// TwinCAT 3 PLC project Simulatore_ASRV
// ProgramVersion: 3.1.4023.0
// libraries:
//   Tc2_Standard, * (Beckhoff Automation GmbH)
//   Tc2_System, * (Beckhoff Automation GmbH)
//   Tc2_Utilities, * (Beckhoff Automation GmbH)
//   Tc3_Module, * (Beckhoff Automation GmbH)
//   VisuDialogs, * (System)
//   VisuSymbols,3.5.10.0,System
// project tree:
//   DUTs/ ASRV.TcDUT, RX_CMD_PC.TcDUT, Comando_PC.TcDUT, CMD_PC.TcDUT, RX_MIS_PC.TcDUT, MIS_PC.TcDUT, Stato_ASRV.TcDUT, Stato_Aux_ASRV.TcDUT, Comandi.TcDUT, Step_PC.TcDUT, RX_Step_PC.TcDUT, TX_STA_ASRV.TcDUT, STA_ASRV.TcDUT
//   / Gestore di visualizzazione.TcVMO (not stored), GlobalTextList.TcGTLO, PlcTask.TcTTO, VISU_TASK.TcTTO
//   GVLs/ Var_Globali.TcGVL
//   POUs/ Check_Com_PC.TcPOU, FB_ClassASRV.TcPOU, FB_File_Write.TcPOU, FB_File_Read.TcPOU, MAIN.TcPOU, Simula_Compila_Mis.TcPOU, Simula_Compila_Sta.TcPOU, Reset_Mis.TcPOU, Simula_Run_Mis.TcPOU, FB_Test_XXX.TcPOU, Trasf_Sta_TxSta.TcPOU, Trasf_RxMiss_Miss.TcPOU, Trasf_RxCmd_Cmd.TcPOU
//   VISUs/ Visualization.TcVIS
// real-time tasks:
//   TASK PlcTask: cycle T#10ms, priority 6, ADS port 350
//   TASK VISU_TASK: cycle T#100000us, priority 8, ADS port 351

CONFIGURATION Simulatore_ASRV
    RESOURCE PLC ON TwinCAT3
        TASK PlcTask(INTERVAL := T#10ms, PRIORITY := 6);
        TASK VISU_TASK(INTERVAL := T#100000us, PRIORITY := 8);
        PROGRAM MAIN WITH PlcTask : MAIN;
        PROGRAM VisuElems_Visu_Prg WITH VISU_TASK : VisuElems.Visu_Prg;
    END_RESOURCE
END_CONFIGURATION

// ---- DUTs/ASRV.TcDUT
TYPE ASRV :
STRUCT
	ASRV_MIS 	: MIS_PC;		// missione da PC
	ASRV_CMD	: CMD_PC;		// comandi da PC
	ASRV_STA	: STA_ASRV;		// stato ASRV
	ASRV_num 	: UINT;			// numero ASRV
END_STRUCT
END_TYPE

// ---- DUTs/RX_CMD_PC.TcDUT
TYPE RX_CMD_PC :
STRUCT
	WatchDog_PC        : UINT;  		// Check di rete (PC++, ASRV pareggia) 
	Start_Miss_PC      : UINT;			// Start Missione da PC. Start=1, azzera appena Stato_Miss_ASRV=1
	End_Miss_PC        : UINT;			// Fine Missione da PC. End=1, appena Stato_Miss_ASRV=2 o per forz.PC
	Pintend_PC         : UINT;			// Nodo intermedio missione = Nodo semaforo di stop
	New_Pos_PC         : UINT;			// Nodo assegnato da PC a ASRV
	Comando_PC         : WORD;			// Word (16 bit) --> struttura Comando PC (16 byte)			
END_STRUCT
END_TYPE

// ---- DUTs/Comando_PC.TcDUT
TYPE Comando_PC :
STRUCT
	Stop    : BOOL; 	// Arresta ASRV immediatamente 
	Aux1	: BOOL;			
	Aux2	: BOOL;			
	Aux3	: BOOL;			
	Aux4	: BOOL;			
	Aux5	: BOOL;			
	Aux6	: BOOL;			
	Aux7	: BOOL;			
	Aux8	: BOOL;			
	Aux9	: BOOL;			
	Aux10	: BOOL;			
	Aux11	: BOOL;			
	Aux12	: BOOL;			
	Aux13	: BOOL;			
	Aux14	: BOOL;			
	Aux15	: BOOL;			
 END_STRUCT
END_TYPE

// ---- DUTs/CMD_PC.TcDUT
TYPE CMD_PC :
STRUCT
	WatchDog_PC        : UINT;  		// Check di rete (ASRV++, PC pareggia) 
	Start_Miss_PC      : UINT;			// Start Missione da PC. Start=1, azzera appena Stato_Miss_ASRV=1
	End_Miss_PC        : UINT;			// Fine Missione da PC. End=1, appena Stato_Miss_ASRV=2 o per forz.PC
	Pintend_PC         : UINT;			// Nodo intermedio missione = Nodo semaforo di stop
	New_Pos_PC         : UINT;			// Nodo assegnato da PC a ASRV
	Comando_PC         : Comando_PC;	// struttura Comando PC			
END_STRUCT
END_TYPE

// ---- DUTs/RX_MIS_PC.TcDUT
TYPE RX_MIS_PC :
STRUCT
	Step_PC       : ARRAY[0..MAX_STEP_MISS] OF RX_Step_PC; // Word ==> step programma 0..500
	Tot_step_PC	  : UINT;						 // Numero di steps della missione
	Pstart_PC     : UINT;						 // Nodo iniziale missione (=Nodo attuale ASRV)
	Pend_PC       : UINT;						 // Nodo fine missione (eventuale di carico/scarico)
	Typ_car_PC    : UINT;						 // Tipo di stabilità carico (0 massima, 9 minima)
	MisFree1      : UINT;
	MisFree2      : UINT;
	MisFree3      : UINT;
END_STRUCT
END_TYPE

// ---- DUTs/MIS_PC.TcDUT
TYPE MIS_PC :
STRUCT
	Step_PC       : ARRAY[0..MAX_STEP_MISS] OF Step_PC;	// Array step programma  (0..500)
	Tot_step_PC	  : UINT;						// Numero di steps della missione
	Pstart_PC     : UINT;						// Nodo iniziale missione (=Nodo attuale ASRV)
	Pend_PC       : UINT;						// Nodo fine missione (eventuale di carico/scarico)
	Typ_car_PC    : UINT;						// Tipo di stabilità carico (0 massima, 9 minima)
	MisFree1      : UINT;
	MisFree2      : UINT;
	MisFree3      : UINT;
END_STRUCT
END_TYPE

// ---- DUTs/Stato_ASRV.TcDUT
TYPE Stato_ASRV :
STRUCT
	In_Mov_X      : BOOL;	// In movimento su asse X (orizz)
	In_Mov_Y      : BOOL;	// In movimento su asse Y (vert)
	In_Mov_Av     : BOOL;	// In movimento direzione +
	In_Mov_Ind    : BOOL;	// In movimento direzione -
	In_Allarme    : BOOL;	// In allarme
	Ok_Prog       : BOOL;	// Pronto a ricevere Missione
	In_Automatico : BOOL;	// In Automatico
	In_Manuale    : BOOL;	// In Manuale	
	Su_Nodo       : BOOL;	// Posizionato su Nodo
	Carico        : BOOL;	// Pallet a bordo
	PosSoll_0     : BOOL;	// Codifica pos. alzata pallet bit.0
	PosSoll_1     : BOOL;	// Codifica pos. alzata pallet bit.1
	Rich_Reset    : BOOL;	// Richiede reset missione a Supervisore
	Aux13         : BOOL;
	Aux14         : BOOL;
	Aux15         : BOOL;
END_STRUCT
END_TYPE

// ---- DUTs/Stato_Aux_ASRV.TcDUT
TYPE Stato_Aux_ASRV :
STRUCT
	Fermo_in_X    : BOOL;	// Fermo su asse X (orizz)
	Fermo_in_Y    : BOOL;	// Fermo su asse Y (vert)
	Rotaz_in_X    : BOOL;	// In rotazione verso asse X
	Rotaz_in_y    : BOOL;	// In rotazione verso asse X
	In_Ricarica   : BOOL;	// In ricarica batteria
	In_Sost_Batt  : BOOL;	// In sostituzione batteria
	In_Manutenz   : BOOL;	// In manutenzione
	Aux7          : BOOL;		
	Aux8          : BOOL;	
	Aux9          : BOOL;	
	Aux10         : BOOL;	
	Aux11         : BOOL;	
	Aux12         : BOOL;	
	Aux13         : BOOL;
	Aux14         : BOOL;
	Aux15         : BOOL;
END_STRUCT
END_TYPE

// ---- DUTs/Comandi.TcDUT
TYPE Comandi :
STRUCT
	In_Mov_X    : BOOL;		// Muovi su asse X
	In_Mov_Y    : BOOL;		// Muovi su asse Y
	In_Mov_Av   : BOOL;		// Muovi direzione +
	In_Mov_Ind  : BOOL;		// Muovi direzione -
	CarSoll_0   : BOOL;		// Carica pallet (codice alza pallet bit 0)
	CarSoll_1   : BOOL;		// Carica pallet (codice alza pallet bit 1)
	Scarica     : BOOL;		// Scarica pallet
	Lenta       : BOOL;		// Muovi in lenta
	End         : BOOL;		// Fine Missione (ultimo step)
	Aux9		: BOOL;		
	Aux10		: BOOL;	
	Aux11		: BOOL;
	Aux12		: BOOL;
	Aux13		: BOOL;
	Aux14		: BOOL;
	Aux15		: BOOL;
END_STRUCT
END_TYPE

// ---- DUTs/Step_PC.TcDUT
TYPE Step_PC :
STRUCT
	Comandi      : Comandi;
	ps		     : UINT;		// Nodo da raggiungere nello step
	dist	     : UINT;		// Distanza del Nodo da raggiungere (in cm)
	rall	     : UINT;		// Rallentamento speccifico nello Step
	CmFree1		 : UINT;		
	CmFree2		 : UINT;		
	CmFree3		 : UINT;		
END_STRUCT
END_TYPE

// ---- DUTs/RX_Step_PC.TcDUT
TYPE RX_Step_PC :
STRUCT
	Comandi      : WORD;		// Word (16 bit) ==> comandi (16 byte)
	ps		     : UINT;		// Nodo da raggiungere nello step
	dist	     : UINT;		// Distanza del Nodo da raggiungere (in cm)
	rall	     : UINT;		// Rallentamento specifico nello Step
	CmFree1		 : UINT;		
	CmFree2		 : UINT;		
	CmFree3		 : UINT;		
END_STRUCT
END_TYPE

// ---- DUTs/TX_STA_ASRV.TcDUT
TYPE TX_STA_ASRV :
STRUCT
	WatchDog_ASRV        : UINT;  			// Check di rete (ASRV++, PC pareggia) 
	Pos_ASRV             : UINT; 	    	// Nodo attuale ASRV
	Stato_Miss_ASRV      : UINT;			// Stato Missione ASRV (0=idle, 1=attiva, 2=completa)
	Stato_ASRV           : WORD;		    // Word (16 bit) ==> struct Stato_ASRV (16 byte)
	Stato_Aux_ASRV 	     : WORD;		 	// Word (16 bit) ==> struct Stato_Aux_ASRV (16 byte)
	ptr_step_ASRV	     : UINT;			// Puntatore passo programma (in esecuzione)
	offset_da_nodo_ASRV  : UINT;			// distanza da ultimo Nodo (in cm)
	Allarmi_1_ASRV       : WORD;			// allarmi ASRV word 1
	Allarmi_2_ASRV       : WORD;			// allarmi ASRV word 2
	Allarmi_3_ASRV       : WORD;			// allarmi ASRV word 3
	Allarmi_4_ASRV       : WORD;			// allarmi ASRV word 4
	Perc_Batteria_ASRV   : UINT;			// % batteria ASRV (0-100)
	Peso_Teorico_ASRV    : UINT;			// peso a bordo da celle di carico
	StFree1              : UINT;			
	StFree2              : UINT;			
	StFree3              : UINT;			
	StFree4              : UINT;			
	StFree5              : UINT;			
 END_STRUCT
END_TYPE

// ---- DUTs/STA_ASRV.TcDUT
TYPE STA_ASRV :
STRUCT
	WatchDog_ASRV        : UINT;  			// Check di rete (ASRV++, PC pareggia) 
	Pos_ASRV             : UINT; 	    	// Nodo attuale ASRV
	Stato_Miss_ASRV      : UINT;			// Stato Missione ASRV (0=idle, 1=attiva, 2=completa)
	Stato_ASRV           : Stato_ASRV;		// struct Stato_ASRV
	Stato_Aux_ASRV 	     : Stato_Aux_ASRV;	// struct Stato_Aux_ASRV
	ptr_step_ASRV	     : UINT;			// Puntatore passo programma (in esecuzione)
	offset_da_nodo_ASRV  : UINT;			// distanza da ultimo Nodo (in cm)
	Allarmi_1_ASRV       : WORD;			// allarmi ASRV word 1
	Allarmi_2_ASRV       : WORD;			// allarmi ASRV word 2
	Allarmi_3_ASRV       : WORD;			// allarmi ASRV word 3
	Allarmi_4_ASRV       : WORD;			// allarmi ASRV word 4
	Perc_Batteria_ASRV   : UINT;			// % batteria ASRV (0-100)
	Peso_Teorico_ASRV    : UINT;			// peso a bordo da celle di carico
	StFree1              : UINT;			
	StFree2              : UINT;			
	StFree3              : UINT;			
	StFree4              : UINT;			
	StFree5              : UINT;			
 END_STRUCT
END_TYPE

// ---- GVLs/Var_Globali.TcGVL
//{attribute 'qualified_only'}
VAR_GLOBAL PERSISTENT
	//--------------------- var globali
	nNumAsrv  : UINT:=1;		// Numero ASRV		
	sSta      : STA_ASRV;		// Stato ASRV (tx a PC)
	sCmd      : CMD_PC;			// Comando ASRV (rx da PC)
	sMis	  : MIS_PC;			// Missione ASRV (rx da PC)
	//--------------------- classe ASRV
	fbClassAsrv	: FB_ClassASRV();	// Classe ASRV
	//--------------------- per visualizzazione 
	sLastStep : Step_PC;		// ultimo Step elaborato	
	//-------------------- Test #####
	nSimCmSpost : UINT :=1 ;	// Siumlazione: Vel. cm 1/10sec spostamento Veloce
	nRappVelLen : UINT :=10;	// Rapporto Vel su Lenta (10 = lenta 1/10 della veloce)	 
	fCmSpostAtt : REAL :=0;		// Velocità spostam. attuale
		
END_VAR

VAR_GLOBAL
	//--------------------- buffer comunicazione
	sTxSta    : TX_STA_ASRV;	// Tx a PC Stato ASRV
	sRxCmd    : RX_CMD_PC;		// Rx da PC Comandi per ASRV
	sRxMis	  : RX_MIS_PC;		// Rx da PC Missione per ASRV
    Old_WatchDog_PC   : UINT;   // Check di rete (PC++, ASRV pareggia) 
	bResetMis : BOOL := FALSE;	// Flag per reset Missione a bordo ASRV

	//-------------------- Test #####
	bSimulaMis 	: BOOL := FALSE;  		// Trigger elaborazione simula missione 	-> compila "sMis"
	bSimulaSta	: BOOL := FALSE;  		// Trigger elaborazione compila Stato   	-> compila "sSta"
	bSimulaRun	: BOOL := TRUE;  		// Abilita Simulazione avanzamento missione -> compila "sSta"
	bSimulaStep	: BOOL := FALSE;  		// Abilita Simulazione avanzamento Step by Step (alla fine di ogni Step toglie il bSimulaRun)
	bSimTrigRun	: BOOL := FALSE;  		// Trigger elaborazione Simulazione avanzamento missione 
	fbTSimRun   : TON := (PT:=T_RUN_MIS);// Timer Simulazione avanzamento missione
	uCntSimRun	: LINT :=0;				// Cnt elaborazioni Simulazione Run
	bSimRunNew	: BOOL := FALSE;		// Flag Step concluso: inizio nuovo 
	bFilpFlopCycle: BOOL := FALSE;		// bistabile ciclo
	bCambioDir	: BOOL := FALSE;		// Indica Step di movimento con cambio direzione
	fbTCambioDir: TON := (PT:=T#2S);	// Tmr. per cambio direzione X/Y
	bCarScar	: BOOL := FALSE;		// Indica Step di carico/scarico
	fbTCarScar  : TON := (PT:=T#3S);	// Tmr. per carico/scarico
	//-------------------- dimensione buffers
	nDimSTA   : UINT :=0;
	nDimCMD   : UINT :=0;
	nDimMIS   : UINT :=0;
	nDimRxSTA : UINT :=0;
	nDimRxCMD : UINT :=0;
	nDimRxMIS : UINT :=0;
	//------------------- comunicazione
	bErrComPc  : BOOL := FALSE;
	nErrComPC  : UINT :=0;						// Flag Errore comunicazione con PC	
	fbToutCom  : TON := (PT:=T_OUT_COMUNICAZ);	// Timeout comunicazione con PC
	fbTPresCmd : TON := (PT:=T_PRES_CMD);		// Rit. presenza nuovo CMD su Buffer Rx PC
	fbTPresMis : TON := (PT:=T_PRES_MIS);		// Rit. presenza nuova MIS su Buffer Rx PC
	
	//------------------ Utilizzati per Test passaggio strutture a FB
	TestMis_XXX      : MIS_PC;						
	fbTestMis_XXX    : FB_Test_XXX;	

END_VAR

VAR_GLOBAL CONSTANT
	RAP_VEL_LENTA	  : UINT := 10;		// Rapporto veloce su lenta (spostamento ASRV) 	
	MAX_STEP_MISS     : UINT := 500;	// Nr. massimo di Step Missione	
	PESO_FITTIZIO_SIM : UINT := 900;	// Kg pallet	
	T_OUT_COMUNICAZ	  : TIME := T#5S;	// Timeout coumunicazione PC/ASRV
	T_RUN_MIS	  	  : TIME := T#100MS;// Tmr clock run missione
	T_PRES_CMD	  	  : TIME := T#200MS;// Tmr sicurezza pres. Nuovo comando da PC per ASRV
	T_PRES_MIS	  	  : TIME := T#1S;	// Tmr sicurezza pres. Nuova missione da PC per ASRV
END_VAR

// ---- POUs/MAIN.TcPOU
PROGRAM MAIN
VAR 
	bError 		: BOOL := FALSE;
	bByPassPC 	: BOOL := FALSE;	// Aux per test senza PC	
	sX			: ASRV;				// appoggio struct ASRV
	bPresRxMis	: BOOL :=FALSE;		// flag presenza dati su buffer Rx
	bPresRxCmd	: BOOL :=FALSE;		// flag presenza dati su buffer Rx

	//-------------------- scrittura / lettura file
	nAux		: UINT := 0;
	sPath		: STRING;
	sMessagg	: STRING;
	fbFileWrite : FB_File_Write;
	bWrite		: BOOL	:=FALSE;	// Trigger write	
	bWriteOk	: BOOL	:=FALSE;	// write Ok
	bWriteErr	: BOOL	:=FALSE;	// write Err	
	fbFileRead  : FB_File_Read;
	bRead		: BOOL	:=FALSE;	// Trigger Read	
	bReadOk		: BOOL	:=FALSE;	// Read Ok
	bReadErr	: BOOL	:=FALSE;	// Read Err	
	
END_VAR


//@@@@@@
//---------------------------------------------------
// test passaggio parametri a FB
//---------------------------------------------------
TestMis_XXX.Tot_step_PC:=10;
fbTestMis_XXX.TestMisPOINT_XXX := ADR(TestMis_XXX);		// Passaggio Tramite Pointer
fbTestMis_XXX.TestMisREFER_XXX := ADR(TestMis_XXX);		// Passaggio Tramite Reference
fbTestMis_XXX();
//@@@@@@

//----------------------------------------------------
// Check dimensione strutture (per confronto con PC)
//----------------------------------------------------
nDimRxCMD 	:= SIZEOF(RX_CMD_PC); 	// check dimensione
nDimRxMIS 	:= SIZEOF(RX_MIS_PC); 	// check dimensione
nDimRxSTA 	:= SIZEOF(TX_STA_ASRV); // check dimensione
nDimCMD 	:= SIZEOF(CMD_PC); 		// check dimensione
nDimMIS 	:= SIZEOF(MIS_PC); 		// check dimensione
nDimSTA 	:= SIZEOF(STA_ASRV); 	// check dimensione

bFilpFlopCycle := NOT bFilpFlopCycle;

//#####	
//------------------------------------------------------
// Lettura numero ASRV da File 'C:\ASRV\ASRV_NUM.TXT'
// se errore assegna numero ASRV = 99
//------------------------------------------------------
sPath := 'C:\ASRV\ASRV_NUM.TXT';
IF _TaskInfo[1].FirstCycle = TRUE THEN		// 1° ciclo scansione PLC
	bRead := TRUE;
	nNumAsrv := 99;							// default se manca file o errore lettura
END_IF
// Lettura -> "nNumAsrv"
fbFileRead(bStart:=bRead, sFileName:=sPath, sMess:=sMessagg, 	// nome file + messaggio
		    nModeOpen:=FOPEN_MODEREAD OR FOPEN_MODETEXT,		// apertura, testo		
            bOperaz_Ok:=bReadOk, bOperaz_Err:=bReadErr);		// risultato
IF bReadOk = TRUE THEN
	nAux := TO_UINT(sMessagg);
	IF nAux <1 OR nAux>20 THEN
		nAux 	 :=99;						// default se manca file o errore lettura
		bReadErr := TRUE;
		bReadOk  := FALSE;
	END_IF
	nNumAsrv :=nAux;
END_IF
IF bReadErr = TRUE THEN
	sMessagg := TO_STRING(nNumAsrv);
	bWrite := TRUE;
END_IF
bReadOk  := FALSE;
bReadErr  := FALSE;
// Scrittura
// (creazione file se errore lettura e scrive 99) 
fbFileWrite(bStart:=bWrite, sFileName:=sPath, sMess:=sMessagg, 	// nome file + messaggio
		    nModeOpen:=FOPEN_MODEWRITE OR FOPEN_MODETEXT,		// sovrascrittura, testo		
            bOperaz_Ok:=bWriteOk, bOperaz_Err:=bWriteErr);		// risultato
IF bWriteErr = TRUE OR bWriteOk = TRUE THEN
	bWriteOk  := FALSE;
	bWriteErr  := FALSE;
END_IF
//#####	


//----------------------------------------------------------------
// Check comunicazione Ok con PC  e pareggia WatchDog Stato ASRV
//----------------------------------------------------------------
nErrComPC := 1;
fbClassAsrv.Get_sAsrv(auxAsrv:=sX);//##>>				// "sAsrv" >> "sX"
sX.ASRV_num := nNumAsrv;								// Assegna Nr. ASRV
Check_Com_PC(nWatchDogPC:=sRxCmd.WatchDog_PC, 
             nWatchDogASRV:=sX.ASRV_STA.WatchDog_ASRV,	
			 fbTout:=fbToutCom,
			 nErroreCom:=nErrComPC ); 
fbClassAsrv.Set_sAsrv(auxAsrv:=sX);//##<<				// "sAsrv" << "sX"

//-------------------------------------------------------------------------
// === RX da PC (CMD,MIS) === 
// Rit. presenza nuovi dati su Buffer Rx PC.
// Essendo il PLC passivo nella comunicazione, per capire se è presente
// un nuovo dato nei buffer RX "sRxCmd" e "sRxMis", controlliamo che il valore di 
// 	  	"sRxCmd.WatchDog_PC" > 0 && <> "Old_WatchDog_PC" (sempre)
// 	  	"sRxMis.Tot_step_PC" > 0	(sempre)
// Se Si, facciamo decorrere un tempo (sicurezza buffer completo) e quindi
// acquisiamo il dato nel buffer di lavoro:
//  	"sRxCmd" >> "sCmd"
//  	"sRxMis" >> "sMis"
// Successivamente aggiorniamo il valore di:
// 	  	"Old_WatchDog_PC" := "sRxCmd.WatchDog_PC" 
// 	  	"sRxMis.Tot_step_PC" :=0
// La prossima lettura compilerà nuovamente i buffer Rx con valori >0
//-------------------------------------------------------------------------
bPresRxCmd := FALSE;
bPresRxMis := FALSE;
IF nErrComPC = 0 OR bByPassPC THEN
	IF sRxCmd.WatchDog_PC>0 AND sRxCmd.WatchDog_PC<>Old_WatchDog_PC THEN
		bPresRxCmd := TRUE;
	END_IF
	IF sRxMis.Tot_step_PC>0 THEN
		bPresRxMis := TRUE;
	END_IF
END_IF	
fbTPresCmd( IN:=bPresRxCmd );	// Tmr presenza nuovi dati in Buffer Rx "sRxCmd" 	
fbTPresMis( IN:=bPresRxMis );	// Tmr presenza nuovi dati in Buffer Rx "sRxMis" 

//-------------------------------------------------------
// Trasferisce "sRxCmd" e "sRxMis" ricevuti da PC 
// su Var.Globali "sCmd" e "sMis", dopo un tmr di sicurezza 
// presenza dati, solo se non errore di comunicazione
//-------------------------------------------------------

IF nErrComPC = 0 OR bByPassPC THEN
	//------------------------------------------------------
	// Trasferisce "sRxCmd" e "sRxMis" ricevuti da PC 
	// "sRxCmd" >> "sCmd" (scompatta le Word)
	// "sRxMis" >> "sMis" (scompatta le Word)
	// "sMis" e "sCmd" vengono compilate impulsivmanete 
	// dopo un tempo di pres.dati in buffer Rx.
	//------------------------------------------------------
	IF fbTPresMis.Q = TRUE THEN								// Tmr pres.nuovo buffer missione scaduto
		Trasf_RxMiss_Miss( auxRxMis:=sRxMis, auxMis:=sMis );// "sRxMis" --> "sMis"  
	END_IF
	IF fbTPresCmd.Q = TRUE THEN								// Tmr pres.nuovo buffer comando scaduto 
		Old_WatchDog_PC := sRxCmd.WatchDog_PC;				// aggiorna "Old_WatchDog_PC"
		Trasf_RxCmd_Cmd( auxRxCmd:=sRxCmd , auxCmd:=sCmd );	// "sRxCmd" --> "sCmd"  
		//------------------------------------------------
		// Rx Nuova Posizione da PC --> Pos_ASRV
		//------------------------------------------------
		fbClassAsrv.Get_sAsrv(auxAsrv:=sX);//##>>				// "sAsrv" >> "sX"
		IF sCmd.New_Pos_PC > 0 AND sX.ASRV_STA.Stato_Miss_ASRV=0 THEN 
			sX.ASRV_STA.Pos_ASRV := sCmd.New_Pos_PC;
			sX.ASRV_STA.offset_da_nodo_ASRV := 0;
			sX.ASRV_STA.Stato_ASRV.Su_Nodo := TRUE;
			//-------------------------------- memorizza stop su direzione X,Y
			IF sX.ASRV_STA.Stato_ASRV.In_Mov_X = TRUE THEN
				sX.ASRV_STA.Stato_Aux_ASRV.Fermo_in_X := TRUE;	
			END_IF
			IF sX.ASRV_STA.Stato_ASRV.In_Mov_Y = TRUE THEN
				sX.ASRV_STA.Stato_Aux_ASRV.Fermo_in_Y := TRUE;	
			END_IF
			sX.ASRV_STA.Stato_ASRV.In_Mov_Av := FALSE;
			sX.ASRV_STA.Stato_ASRV.In_Mov_Ind := FALSE;
			sX.ASRV_STA.Stato_ASRV.In_Mov_X := FALSE;
			sX.ASRV_STA.Stato_ASRV.In_Mov_Y := FALSE;
		END_IF
		fbClassAsrv.Set_sAsrv(auxAsrv:=sX);//##<<				// "sAsrv" << "sX"
	END_IF
	//------------------------------------------------------
	// Aggiorna Classe "sAsrv" con "sCmd" e "sMis" Rx da PC
	// Se non errore di comunicazione
	//------------------------------------------------------
	fbClassAsrv.Aggiorna_CMD_da_PC(auxCmd := sCmd);			// "sCmd" >> "sAsrv"
	fbClassAsrv.Aggiorna_MIS_da_PC(auxMis := sMis);  		// "sMis" >> "sAsrv"
END_IF			 

//################################################ Gestione
//################################################ Gestione
//################################################ Gestione

//-------------------------------------------------
// Forza Reset Missione
// Flag attivato da PC "End_Mis_PC=1" o forzato PLC
//-------------------------------------------------
IF bResetMis=TRUE THEN												
	bResetMis :=FALSE;
	bError := fbClassAsrv.Azzera_MIS();							// Reset Missione >> azzera ASRV 1 
	//-------------------------------------
	// Azzera var.globale "sMis" 
	//-------------------------------------
	fbClassAsrv.Get_sAsrv(auxAsrv:=sX);//##>>					// "sAsrv" >> "sX"
	Reset_Mis(auxMis := sMis, auxSta:= sX.ASRV_STA);		    // Reset "sMis" + aggiorna stato sX (ptr step, stato_miss)
	sRxMis.Tot_step_PC := 0;									// Reset "sRxMis.Tot_step_PC" (buffer Rx da PC - dovrebbe essere già 0)
	fbClassAsrv.Set_sAsrv(auxAsrv:=sX);//##<<					// "sAsrv" << "sX"
END_IF


//############ Simulazione ##############
//############ Simulazione ##############
//------------------------------------------
// Simula cambio Stato "sAsrv" - STA
// Flag forzato PLC 
// Nella funzione possiamo impostare lo  
// stato ASRV come vogliamo
//------------------------------------------
IF bSimulaSta=TRUE THEN
	bSimulaSta :=FALSE;
	//-------------------compila "sAsrv" - STA (Stato)
	fbClassAsrv.Get_sAsrv(auxAsrv:=sX);//##>>			// "sAsrv" >> "sX" 
	Simula_Compila_Sta( nNodo:=143, bCarico:=FALSE, sX.ASRV_STA ); 	// Compila Stato >> "sX"
	fbClassAsrv.Set_sAsrv(auxAsrv:=sX);//##<<			// "sAsrv" << "sX"
END_IF
//-----------------------------------------------------
// Simula Nuova Missione da PC "sMis" -> "sAsrv" - MIS
// Flag forzato PLC 
// Nella funzione possiamo impostare la  
// missione ASRV come vogliamo
//-----------------------------------------------------
IF bSimulaMis=TRUE THEN
	bSimulaMis :=FALSE;
	bError := fbClassAsrv.Azzera_MIS();					// Reset Mis >> "sAsrv"
	//-------------------compila "sMis"
	Simula_Compila_Mis( auxMis := sMis );				// compila Missione >> "sMis" (da PC)
    fbClassAsrv.Aggiorna_MIS_da_PC(auxMis := sMis);		// "sMis" >> "sAsrv"
END_IF
//-----------------------------------------------------------------
// Simula Run Missione (con Missione attiva)
// L'elaborazione degli Step modifica lo stato "sAsrv" - STA
//-----------------------------------------------------------------
fbClassAsrv.Get_sAsrv(auxAsrv:=sX);//##>>			// "sAsrv" >> "sX" 
Simula_Run_Mis( auxSta:=sX.ASRV_STA, auxMis:=sX.ASRV_MIS, auxCmd:= sX.ASRV_CMD, bError=>bError ); 
fbClassAsrv.Set_sAsrv(auxAsrv:=sX);//##<<			// "sAsrv" << "sX"

//############ Simulazione ##############
//############ Simulazione ##############


//------------------------------------------
// Gestione Flag Start/End Missione
// Start / End sempre da "Cmd" PC
//------------------------------------------
fbClassAsrv.Get_sAsrv(auxAsrv:=sX);//##>>				// "sAsrv" >> "sX"
//----------------------------------------
// Start missione da PC -> Start ASRV=1
// Dopo aver ricevuto la missione si attende 
// che PC attivi "sCmd.Start_Mis_PC=1"
//----------------------------------------
IF sX.ASRV_CMD.Start_Miss_PC = 1 THEN
	sX.ASRV_STA.Stato_Miss_ASRV :=1; 					// Stato Miss ASRV  = 1
	sX.ASRV_STA.Stato_ASRV.Ok_Prog := FALSE;			// Stato Ok_Prog = 0
END_IF
//-----------------------------------------------------
// End missione da PC -> Start ASRV=0 + Reset missione
// Dopo aver concluso la missione si attende 
// che PC attivi "sCmd.End_Mis_PC=1"
//-----------------------------------------------------
IF sX.ASRV_CMD.End_Miss_PC = 1 THEN
	sX.ASRV_STA.Stato_Miss_ASRV :=0;					// Stato Miss ASRV  = 0
	sX.ASRV_STA.Stato_ASRV.Ok_Prog := TRUE;				// Stato Ok_Prog = 1
	bResetMis := TRUE;									// flag x Reset Missione
END_IF
fbClassAsrv.Set_sAsrv(auxAsrv:=sX);//##<<				// "sAsrv" << "sX"

//################################################ Gestione
//################################################ Gestione
//################################################ Gestione



//--------------------------------------------------
// === TX a PC (STA) === 
// Aggiorna STA da Tx a PC con Classe ASRV 
//--------------------------------------------------
bError := fbClassAsrv.Aggiorna_STA_a_PC(auxSta := sSta);// trasf. "sAsrv" >> "sSta" (stato per PC)	
//------------------------------------------------------
// Prepara Stato ASRV per Tx a PC (+ compatta Word)
//------------------------------------------------------
Trasf_Sta_TxSta( auxSta:=sSta, auxTxSta:=sTxSta );		// Stato "sSta" >> "sTxSta" (STATO TX a PC)

END_PROGRAM

// ---- POUs/FB_File_Write.TcPOU
FUNCTION_BLOCK PUBLIC FB_File_Write
VAR_INPUT
	bStart  	: REFERENCE TO BOOL;		// Flag operazione
	sFileName 	: REFERENCE TO STRING;		// Nome file + path
	sMess   	: REFERENCE TO STRING;		// messaggio / read / write
	nModeOpen  	: DWORD;					// modalità di apertura
	bOperaz_Ok	: REFERENCE TO BOOL;		// risultato Ok			
	bOperaz_Err : REFERENCE TO BOOL;		// risultato Err
END_VAR
VAR
	// Istanza gestione file 
	fbFileOpen  : FB_FileOpen;		
	fbFileClose : FB_FileClose;
	fbFilePuts  : FB_FilePuts;
	fbFileGets  : FB_FileGets;
	eState 		: (IDLE, OPEN_TRIGGER, OPEN, WRITE_TRIGGER, WRITE, CLOSE_TRIGGER, CLOSE, ERROR, OK );
	bError		: BOOL := FALSE;
END_VAR

IF bStart = TRUE THEN
	eState := OPEN_TRIGGER;
	bStart := FALSE;
	bOperaz_Ok  := FALSE;
	bOperaz_Err := FALSE;
END_IF

CASE eState OF
	IDLE:							// Nulla
	//	
	OPEN_TRIGGER:					// Trigger apertura file
		fbFileOpen(bExecute:=TRUE, sPathName:=sFileName, nMode := nModeOpen);
		eState := OPEN;
	OPEN:							// Attesa file aperto
		fbFileOpen(bExecute:=FALSE);
		IF fbFileOpen.bError THEN
			bError := TRUE;				// -> errore
			eState := ERROR;
		ELSIF NOT fbFileOpen.bBusy AND fbFileOpen.hFile <> 0 THEN
			eState := WRITE_TRIGGER;
		END_IF
	WRITE_TRIGGER:					// Trigger scrittura
		fbFilePuts(bExecute:=TRUE, sLine:=sMess, hFile:=fbFileOpen.hFile );
		eState := WRITE;
	WRITE:							// Attesa scrittura
		fbFilePuts(bExecute:=FALSE);
		IF fbFilePuts.bError THEN
			bError := TRUE;				// -> errore
			eState := CLOSE_TRIGGER;	// -> chiude file
		ELSIF NOT fbFilePuts.bBusy THEN
			eState := CLOSE_TRIGGER;
		END_IF
	CLOSE_TRIGGER:					// Trigger chiusura
		fbFileClose(bExecute:=TRUE, hFile:=fbFileOpen.hFile );
		eState := CLOSE;
	CLOSE:							// Attesa chiusura
		fbFileClose(bExecute:=FALSE);
		IF fbFileClose.bError THEN
			eState := ERROR;
			bError := TRUE;				// -> errore
		ELSIF NOT fbFileClose.bBusy THEN
			IF bError = FALSE THEN
				eState := OK;
			ELSE			
				eState := ERROR;
			END_IF
		END_IF
	OK:								// Fine scrittura Ok
		bOperaz_Ok  := TRUE;
		bOperaz_Err := FALSE;
		eState := IDLE;
	ERROR:							// Fine scrittura Error
		bOperaz_Ok  := FALSE;
		bOperaz_Err := TRUE;
		eState := IDLE;
	
END_CASE

END_FUNCTION_BLOCK

// ---- POUs/FB_File_Read.TcPOU
FUNCTION_BLOCK PUBLIC FB_File_Read
VAR_INPUT
	bStart  	: REFERENCE TO BOOL;		// Flag operazione
	sFileName 	: REFERENCE TO STRING;		// Nome file + path
	sMess   	: REFERENCE TO STRING;		// messaggio / read / write
	nModeOpen  	: DWORD;					// modalità di apertura
	bOperaz_Ok	: REFERENCE TO BOOL;		// risultato Ok			
	bOperaz_Err : REFERENCE TO BOOL;		// risultato Err
END_VAR
VAR
	// Istanza gestione file 
	fbFileOpen  : FB_FileOpen;		
	fbFileClose : FB_FileClose;
	fbFilePuts  : FB_FilePuts;
	fbFileGets  : FB_FileGets;
	eState 		: (IDLE, OPEN_TRIGGER, OPEN, READ_TRIGGER, READ, CLOSE_TRIGGER, CLOSE, ERROR, OK );
	bError		: BOOL := FALSE;
END_VAR

IF bStart = TRUE THEN
	eState := OPEN_TRIGGER;
	bStart := FALSE;
	bOperaz_Ok  := FALSE;
	bOperaz_Err := FALSE;
END_IF

CASE eState OF
	IDLE:							// Nulla
	//	
	OPEN_TRIGGER:					// Trigger apertura file
		fbFileOpen(bExecute:=TRUE, sPathName:=sFileName, nMode := nModeOpen);
		eState := OPEN;
	OPEN:							// Attesa file aperto
		fbFileOpen(bExecute:=FALSE);
		IF fbFileOpen.bError THEN
			bError := TRUE;					// -> errore
			eState := ERROR;
		ELSIF NOT fbFileOpen.bBusy AND fbFileOpen.hFile <> 0 THEN
			eState := READ_TRIGGER;
		END_IF
	READ_TRIGGER:					// Trigger lettura
		//fbFileGets(bExecute:=TRUE, sLine=>sMess, hFile:=fbFileOpen.hFile );
		fbFileGets(bExecute:=TRUE, hFile:=fbFileOpen.hFile );
		eState := READ;
	READ:							// Attesa scrittura
		fbFileGets(bExecute:=FALSE);
		IF fbFileGets.bError THEN
			bError := TRUE;					// -> errore
			eState := CLOSE_TRIGGER;		// -> chiude file
		ELSIF NOT fbFileGets.bBusy THEN
			sMess := fbFileGets.sLine;
			eState := CLOSE_TRIGGER;
		END_IF
	CLOSE_TRIGGER:				// Trigger chiusura
		fbFileClose(bExecute:=TRUE, hFile:=fbFileOpen.hFile );
		eState := CLOSE;
	CLOSE:						// Attesa chiusura
		fbFileClose(bExecute:=FALSE);
		IF fbFileClose.bError THEN
			eState := ERROR;
			bError := TRUE;					// -> errore
		ELSIF NOT fbFileClose.bBusy THEN
			IF bError = FALSE THEN
				eState := OK;
			ELSE			
				eState := ERROR;
			END_IF
		END_IF
	OK:								// Fine lettura Ok
		bOperaz_Ok  := TRUE;
		bOperaz_Err := FALSE;
		eState := IDLE;
	ERROR:							// Fine lettura Error
		bOperaz_Ok  := FALSE;
		bOperaz_Err := TRUE;
		eState := IDLE;
	
END_CASE

END_FUNCTION_BLOCK

// ---- POUs/Check_Com_PC.TcPOU
FUNCTION Check_Com_PC
VAR_INPUT
	nWatchDogPC 	: REFERENCE TO UINT;
	nWatchDogASRV 	: REFERENCE TO UINT;
	nErroreCom 		: REFERENCE TO UINT;
	fbTout 			: REFERENCE TO TON;
END_VAR
VAR 
	bInvWD 			: BOOL; 
END_VAR

//------------------------------------
// Pareggia WatchDog Stato ASRV
// PC Incrementa, ASRV pareggia
//------------------------------------
bInvWD := TRUE;

IF nWatchDogPC <> nWatchDogASRV THEN
	bInvWD := FALSE;
	nWatchDogASRV := nWatchDogPC;
END_IF
//-----------------------------------
// Verifica comunicazione in Errore
//-----------------------------------
fbTout( IN:=bInvWD );
bErrComPc := fbTout.Q;
IF fbTout.Q = TRUE THEN	// Timeout scaduto
	nErroreCom  := 1;
ELSE
	nErroreCom  := 0;
END_IF

END_FUNCTION

// ---- POUs/Trasf_RxMiss_Miss.TcPOU
FUNCTION Trasf_RxMiss_Miss
VAR_INPUT
	auxRxMis : REFERENCE TO RX_MIS_PC;
	auxMis   : REFERENCE TO MIS_PC;
END_VAR
VAR
	ni 			: UINT :=0;
END_VAR

//---------------------------------------------------------------------
// Trasferisce Buffer Missione Rx da PC in Missione ASRV
// Scompatta la Word comandi (16 bit) nella struttura comandi (16 byte)
// MISSIONE Rx --> Missione ASRV
//---------------------------------------------------------------------
// Per evitare di trasferire un dato osoleto, viene sempre azzerato
// il valore di Tot_Step del buffer Rx (non può essere mai 0) 
// in questo modo conpila i dati solo se sono stati effettivamente ricevuti
//---------------------------------------------------------------------------
IF auxRxMis.Tot_step_PC>0 THEN
	auxMis.Tot_step_PC   := auxRxMis.Tot_step_PC;
	auxMis.Pstart_PC     := auxRxMis.Pstart_PC;
	auxMis.Pend_PC       := auxRxMis.Pend_PC;
	auxMis.Typ_car_PC    := auxRxMis.Typ_car_PC;
	auxMis.MisFree1      := auxRxMis.MisFree1;
	auxMis.MisFree2      := auxRxMis.MisFree2;
	auxMis.MisFree3      := auxRxMis.MisFree3;
	//----------- ciclo per tutti gli Step
	FOR ni :=0 TO MAX_STEP_MISS BY 1 DO
		auxMis.Step_PC[ni].ps        := auxRxMis.Step_PC[ni].ps;
		auxMis.Step_PC[ni].dist      := auxRxMis.Step_PC[ni].dist;
		auxMis.Step_PC[ni].rall 	 := auxRxMis.Step_PC[ni].rall;
		auxMis.Step_PC[ni].CmFree1   := auxRxMis.Step_PC[ni].CmFree1;
		auxMis.Step_PC[ni].CmFree2   := auxRxMis.Step_PC[ni].CmFree2;
		auxMis.Step_PC[ni].CmFree3   := auxRxMis.Step_PC[ni].CmFree3;
		//------------------------ Step comandi word -> Bool 
		auxMis.Step_PC[ni].comandi.In_Mov_X   := WORD_TO_BOOL( auxRxMis.Step_PC[ni].comandi AND 1);
		auxMis.Step_PC[ni].comandi.In_Mov_Y   := WORD_TO_BOOL( auxRxMis.Step_PC[ni].comandi AND 2);
		auxMis.Step_PC[ni].comandi.In_Mov_Av  := WORD_TO_BOOL( auxRxMis.Step_PC[ni].comandi AND 4);
		auxMis.Step_PC[ni].comandi.In_Mov_Ind := WORD_TO_BOOL( auxRxMis.Step_PC[ni].comandi AND 8);
		auxMis.Step_PC[ni].comandi.CarSoll_0  := WORD_TO_BOOL( auxRxMis.Step_PC[ni].comandi AND 16);
		auxMis.Step_PC[ni].comandi.CarSoll_1  := WORD_TO_BOOL( auxRxMis.Step_PC[ni].comandi AND 32);
		auxMis.Step_PC[ni].comandi.Scarica    := WORD_TO_BOOL( auxRxMis.Step_PC[ni].comandi AND 64);
		auxMis.Step_PC[ni].comandi.Lenta      := WORD_TO_BOOL( auxRxMis.Step_PC[ni].comandi AND 128);
		auxMis.Step_PC[ni].comandi.End        := WORD_TO_BOOL( auxRxMis.Step_PC[ni].comandi AND 256);
		auxMis.Step_PC[ni].comandi.Aux9       := WORD_TO_BOOL( auxRxMis.Step_PC[ni].comandi AND 512);
		auxMis.Step_PC[ni].comandi.Aux10      := WORD_TO_BOOL( auxRxMis.Step_PC[ni].comandi AND 1024);
		auxMis.Step_PC[ni].comandi.Aux11      := WORD_TO_BOOL( auxRxMis.Step_PC[ni].comandi AND 2048);
		auxMis.Step_PC[ni].comandi.Aux12      := WORD_TO_BOOL( auxRxMis.Step_PC[ni].comandi AND 4096);
		auxMis.Step_PC[ni].comandi.Aux13      := WORD_TO_BOOL( auxRxMis.Step_PC[ni].comandi AND 8192);
		auxMis.Step_PC[ni].comandi.Aux14      := WORD_TO_BOOL( auxRxMis.Step_PC[ni].comandi AND 16384);
		auxMis.Step_PC[ni].comandi.Aux15      := WORD_TO_BOOL( auxRxMis.Step_PC[ni].comandi AND 32768);
	END_FOR
	//----------- azzera Tot_step_PC su buffer RX
	auxRxMis.Tot_step_PC := 0;
END_IF

END_FUNCTION

// ---- POUs/Trasf_RxCmd_Cmd.TcPOU
FUNCTION Trasf_RxCmd_Cmd
VAR_INPUT
	auxRxCmd : REFERENCE TO RX_CMD_PC;
	auxCmd   : REFERENCE TO CMD_PC;
END_VAR
VAR
	ni 			: UINT :=0;
END_VAR


//---------------------------------------------------------------------------
// Trasferisce Buffer Comandi Rx da PC in Comandi ASRV
// Scompatta la Word Comandi_PC (16 bit) nella struttura Comando_PC (16 byte)
// COMANDI Rx --> Comandi ASRV
//---------------------------------------------------------------------------
// Per evitare di trasferire un dato osoleto, viene sempre azzerato
// il valore di WatchDog del buffer Rx (non può essere mai 0) 
// in questo modo conpila i dati solo se sono stati effettivamente ricevuti
//---------------------------------------------------------------------------
IF auxRxCmd.WatchDog_PC>0 THEN
	auxCmd.WatchDog_PC   := auxRxCmd.WatchDog_PC;
	auxCmd.Start_miss_PC := auxRxCmd.Start_miss_PC;
	auxCmd.End_miss_PC   := auxRxCmd.End_miss_PC;
	auxCmd.Pintend_PC    := auxRxCmd.Pintend_PC;
	auxCmd.New_Pos_PC    := auxRxCmd.New_Pos_PC;
	auxCmd.Comando_PC.Stop   := UINT_TO_BOOL( auxRxCmd.Comando_PC AND 1);
	auxCmd.Comando_PC.Aux1   := UINT_TO_BOOL( auxRxCmd.Comando_PC AND 2);
	auxCmd.Comando_PC.Aux2   := UINT_TO_BOOL( auxRxCmd.Comando_PC AND 4);
	auxCmd.Comando_PC.Aux3   := UINT_TO_BOOL( auxRxCmd.Comando_PC AND 8);
	auxCmd.Comando_PC.Aux4   := UINT_TO_BOOL( auxRxCmd.Comando_PC AND 16);
	auxCmd.Comando_PC.Aux5   := UINT_TO_BOOL( auxRxCmd.Comando_PC AND 32);
	auxCmd.Comando_PC.Aux6   := UINT_TO_BOOL( auxRxCmd.Comando_PC AND 64);
	auxCmd.Comando_PC.Aux7   := UINT_TO_BOOL( auxRxCmd.Comando_PC AND 126);
	auxCmd.Comando_PC.Aux8   := UINT_TO_BOOL( auxRxCmd.Comando_PC AND 256);
	auxCmd.Comando_PC.Aux9   := UINT_TO_BOOL( auxRxCmd.Comando_PC AND 512);
	auxCmd.Comando_PC.Aux10  := UINT_TO_BOOL( auxRxCmd.Comando_PC AND 1024);
	auxCmd.Comando_PC.Aux11  := UINT_TO_BOOL( auxRxCmd.Comando_PC AND 2048);
	auxCmd.Comando_PC.Aux12  := UINT_TO_BOOL( auxRxCmd.Comando_PC AND 4096);
	auxCmd.Comando_PC.Aux13  := UINT_TO_BOOL( auxRxCmd.Comando_PC AND 8192);
	auxCmd.Comando_PC.Aux14  := UINT_TO_BOOL( auxRxCmd.Comando_PC AND 16384);
	auxCmd.Comando_PC.Aux15  := UINT_TO_BOOL( auxRxCmd.Comando_PC AND 32768);
END_IF

END_FUNCTION

// ---- POUs/Reset_Mis.TcPOU
FUNCTION Reset_Mis 
VAR_INPUT
	auxMis   : REFERENCE TO MIS_PC;
	auxSta   : REFERENCE TO STA_ASRV;
END_VAR
VAR
	ni	: UINT :=0;
	ndim	: USINT;
END_VAR

//-------------------------------
// Azzera struttura -> MIS  
//-------------------------------
auxMis.Tot_step_PC   := 0;
auxMis.Pstart_PC     := 0;
auxMis.Pend_PC       := 0;
auxMis.Typ_car_PC    := 0;
auxMis.MisFree1      := 0;
auxMis.MisFree2      := 0;
auxMis.MisFree3      := 0;
//------------------------- Reset Step[]
FOR ni :=0 TO MAX_STEP_MISS BY 1 DO
	ndim := TO_USINT(SIZEOF(auxMis.Step_PC[ni]));							// dim. setp (short)
	MEMSET(destAddr:=ADR(auxMis.Step_PC[ni]) , fillByte:=ndim , n:=16#00 );	// max 255 byte!
END_FOR

//----------------------------
// Reset Step programma
//----------------------------
auxSta.ptr_step_ASRV 	:=0;	// Reset puntatori Step
auxSta.Stato_Miss_ASRV 	:=0;	// reset anche Stato Missione (anche se dovrebbe già essere 0)

END_FUNCTION

// ---- POUs/Simula_Compila_Sta.TcPOU
FUNCTION Simula_Compila_Sta 
VAR_INPUT
	nNodo 	: UINT;	// Nodo partenza
	bCarico	: BOOL; // Stato Carico (True)
END_VAR
VAR_INPUT
 	auxSta   : REFERENCE TO STA_ASRV;
END_VAR

//--------------------------------------------------------
// Simula Compilazione Stato Inziale ASRV
// Elaborata impulsivamente  compila stato iniziale ASRV
//--------------------------------------------------------
//---------------------
// Stato inziale ASRV
//---------------------
auxSta.Pos_ASRV := nNodo;	// Nodo partenza;
auxSta.offset_da_nodo_ASRV	:=0;		
auxSta.Stato_Miss_ASRV 		:=0;
auxSta.ptr_step_ASRV		:=0;
auxSta.Perc_Batteria_ASRV	:=100;

auxSta.Stato_ASRV.In_Automatico := TRUE;
auxSta.Stato_ASRV.In_Allarme 	:= FALSE;
auxSta.Stato_ASRV.Ok_Prog		:= TRUE;
auxSta.Stato_ASRV.PosSoll_0		:= FALSE;
auxSta.Stato_ASRV.PosSoll_1		:= FALSE;
auxSta.Stato_ASRV.Carico		:= bCarico;	// Stato carico
IF bCarico = FALSE THEN
	auxSta.Peso_Teorico_ASRV	:= 0;	
END_IF 
auxSta.Stato_ASRV.Su_Nodo		:= TRUE;

END_FUNCTION

// ---- POUs/Simula_Compila_Mis.TcPOU
FUNCTION Simula_Compila_Mis 
VAR_INPUT
	auxMis   : REFERENCE TO MIS_PC;
END_VAR
VAR
	ni	: UINT :=0;
END_VAR

//----------------------------------------------------
// Simula Creazione Missione
// Elaborata impulsivamente compila la missione        
//----------------------------------------------------
auxMis.Pstart_PC		:=143;
auxMis.PEnd_PC			:=175;
auxMis.Typ_car_PC		:=0;		// stabilità max
//------------------ 1
ni := ni + 1;
auxMis.Step_PC[ni].ps 	:= 144;
auxMis.Step_PC[ni].dist := 100;
auxMis.Step_PC[ni].Comandi.In_Mov_Y 	:= TRUE;
auxMis.Step_PC[ni].Comandi.In_Mov_Av 	:= TRUE;
auxMis.Step_PC[ni].Comandi.Lenta 		:= TRUE;	// cambio corsia
//------------------ 2
ni := ni + 1;
auxMis.Step_PC[ni].ps 	:= 154;
auxMis.Step_PC[ni].dist := 100;
auxMis.Step_PC[ni].Comandi.In_Mov_X 	:= TRUE;
auxMis.Step_PC[ni].Comandi.In_Mov_Av 	:= TRUE;
//------------------ 3
ni := ni + 1;
auxMis.Step_PC[ni].ps 	:= 164;
auxMis.Step_PC[ni].dist := 100;
auxMis.Step_PC[ni].Comandi.In_Mov_X 	:= TRUE;
auxMis.Step_PC[ni].Comandi.In_Mov_Av 	:= TRUE;
//------------------ 4
ni := ni + 1;
auxMis.Step_PC[ni].ps 	:= 174;
auxMis.Step_PC[ni].dist := 100;
auxMis.Step_PC[ni].Comandi.In_Mov_X 	:= TRUE;
auxMis.Step_PC[ni].Comandi.In_Mov_Av 	:= TRUE;
//------------------ 5
ni := ni + 1;
auxMis.Step_PC[ni].ps 	:= 175;
auxMis.Step_PC[ni].dist := 100;
auxMis.Step_PC[ni].Comandi.In_Mov_Y 	:= TRUE;
auxMis.Step_PC[ni].Comandi.In_Mov_Av 	:= TRUE;
auxMis.Step_PC[ni].Comandi.Lenta 		:= TRUE;	// cambio corsia
//------------------ 6
ni := ni + 1;
auxMis.Step_PC[ni].ps 	:= 175;
auxMis.Step_PC[ni].dist := 0;						// carico su stesso nodo 175
auxMis.Step_PC[ni].Comandi.CarSoll_0 	:= TRUE;	// carico
//------------------ 7
ni := ni + 1;
auxMis.Step_PC[ni].ps 	:= 175;
auxMis.Step_PC[ni].dist := 0;				// fine miss su stesso nodo 175
auxMis.Step_PC[ni].Comandi.End 	:= TRUE;	// fine miss
//------------------ 
auxMis.Tot_Step_PC	:=ni;					// nr. Tot Step

END_FUNCTION

// ---- POUs/Simula_Run_Mis.TcPOU
FUNCTION Simula_Run_Mis 
VAR_INPUT
	auxSta   : REFERENCE TO STA_ASRV;
	auxMis   : REFERENCE TO MIS_PC;
	auxCmd   : REFERENCE TO CMD_PC;
END_VAR
VAR_OUTPUT
	bError	 : BOOL := FALSE;
END_VAR
VAR
	nStep    : UINT;
	sP	 	 : Step_PC;
	sP_1 	 : Step_PC;			// step successivo
	bStop 	 : BOOL :=FALSE;	
	bRitroso : BOOL :=FALSE;
	fCmVel	 : REAL;
	fCmLen	 : REAL;
	fCmSpost : REAL :=0;
	bCS_Offset : BOOL :=FALSE;	// carico/scarico con offset
END_VAR

//-----------------------------------------
// Tmr sosta per cambio direzione
//-----------------------------------------
fbTCambioDir( IN:=bCambioDir );							// Tmr cambio direzione	
//-----------------------------------------
// Tmr per cambio carico/scarico
//-----------------------------------------
fbTCarScar( IN:=bCarScar );								// Tmr cambio direzione	
//--------------------------------------------------------
// Simula Run Missione ASRV
// Tmr esecuzione x missione
//--------------------------------------------------------
fbTSimRun( IN:=(NOT bSimTrigRun) );						// Tmr esecuzione Run Missione	
bSimTrigRun := fbTSimRun.Q;								// impulso elaborazione
IF bSimTrigRun = FALSE OR bSimulaRun = FALSE THEN		// Se non impulso o non abilitazione simula Run, ritorna
	RETURN;
END_IF
uCntSimRun := uCntSimRun +1;							// Cnt cicli 
fCmVel := TO_REAL(nSimCmSpost);	
fCmLen := fCmVel/ TO_REAL(nRappVelLen);	
//---------------------------------------------------------
// Uscita in attesa di carico/scarico
//---------------------------------------------------------
IF fbTCarScar.Q=TRUE THEN
	bCarSCar:=FALSE;
END_IF
IF bCarSCar=TRUE AND fbTCarScar.Q=FALSE THEN
	RETURN;
END_IF; 

//--------------------------------------------------------
// Verifica Condizioni per non elaborare lo Step
//--------------------------------------------------------
IF auxSta.ptr_step_ASRV >= auxMis.Tot_step_PC OR 
   auxSta.ptr_step_ASRV > MAX_STEP_MISS	      OR 
   	auxSta.Stato_Miss_ASRV <> 1               THEN
   	bError := TRUE;
   RETURN;
END_IF
//---------------------------------------------------------------------
// Se Step attuale = 0 (inizio missione) allora abilita nuovo Step (=1)
//---------------------------------------------------------------------
IF auxSta.ptr_step_ASRV=0 THEN 
	bSimRunNew := TRUE;
END_IF
//---------------------------------------------------
// Se nuovo Step, incrementa puntatore
//---------------------------------------------------
IF bSimRunNew=TRUE THEN 
	auxSta.ptr_step_ASRV := auxSta.ptr_step_ASRV +1;	// Step ++
END_IF	
nStep := auxSta.ptr_step_ASRV;
sP   := auxMis.Step_PC[nStep]; 
sP_1 := auxMis.Step_PC[nStep+1];
sLastStep := sP;				// salva ultimo step x visualizzazione

//------------------------------------------------------------------------------------
// solo x 1° Step !	
// Condizione di ritorno su Nodo Step (avvicinamento a ritroso, decrementa disatnza
// o di allontanamento da Nodo Step (incremento)
//------------------------------------------------------------------------------------
bRitroso := FALSE;							// non ritorno su Nodo ingresso
IF nStep =1 THEN
	IF auxSta.Pos_ASRV = sP.ps THEN				// Se pos.attuale ASRV = Pos.Setp in esecuzione allora ritorno su Nodo precedente
		bRitroso :=TRUE;
	END_IF
END_IF


//--------------------------------------------
// preset stato movimentazione = fermo
//--------------------------------------------
IF auxSta.Stato_ASRV.In_Mov_X = TRUE THEN
	auxSta.Stato_Aux_ASRV.Fermo_in_X := TRUE;	
END_IF
IF auxSta.Stato_ASRV.In_Mov_Y = TRUE THEN
	auxSta.Stato_Aux_ASRV.Fermo_in_Y := TRUE;	
END_IF
auxSta.Stato_ASRV.In_Mov_X   := FALSE;
auxSta.Stato_ASRV.In_Mov_Y   := FALSE;
auxSta.Stato_ASRV.In_Mov_Av  := FALSE;
auxSta.Stato_ASRV.In_Mov_Ind := FALSE;
//----------------------------------------------------
// Se nuovo Step preset posizione, offset=0 + su Nodo 
//----------------------------------------------------
IF bSimRunNew=TRUE THEN 
	
	//§§§§
	IF sP.Comandi.In_Mov_X=FALSE AND sP.Comandi.In_Mov_Y=FALSE THEN
		//--------------------------------------------
		// Passo Carico SENZA offset (non mi sposto)
		//--------------------------------------------
		IF sP.Comandi.CarSoll_0 OR sP.Comandi.CarSoll_1 THEN
			auxSta.Stato_ASRV.Carico := TRUE;
			auxSta.Peso_Teorico_ASRV := PESO_FITTIZIO_SIM;	// fittizio
			bCarSCar:=TRUE;		// Tmr  Carico/Scarico
			//--------------------------------------------------
			// Se abilitato Step, mette in Hold la simulazione
			//--------------------------------------------------
			IF bSimulaStep=TRUE THEN
				bSimulaRun := FALSE;
			END_IF
			RETURN;
		END_IF
		//--------------------------------------------
		// Passo Scarico SENZA offset (non mi sposto)
		//--------------------------------------------
		IF sP.Comandi.Scarica THEN
			auxSta.Stato_ASRV.Carico := FALSE;
			auxSta.Peso_Teorico_ASRV := 0;	
			bCarSCar:=TRUE;		// Tmr  Carico/Scarico
			//--------------------------------------------------
			// Se abilitato Step, mette in Hold la simulazione
			//--------------------------------------------------
			IF bSimulaStep=TRUE THEN
				bSimulaRun := FALSE;
			END_IF
			RETURN;
		END_IF
	END_IF
	//§§§§

	//--------------------------------------------
	// Passo Fine Missione
	//--------------------------------------------
	IF sP.Comandi.End THEN
		auxSta.Stato_Miss_ASRV := 2;
		//--------------------------------------------------
		// Se abilitato Step, mette in Hold la simulazione
		//--------------------------------------------------
		IF bSimulaStep=TRUE THEN
			bSimulaRun := FALSE;
		END_IF
		RETURN;
	END_IF
END_IF
//------------------------------
// reset new step
//------------------------------
bSimRunNew := FALSE;

//--------------------------------------------------
// Passo Spostamento + Carico/Scarico con offset
//--------------------------------------------------
IF sP.Comandi.In_Mov_X OR sP.Comandi.In_Mov_Y THEN
	//----------------------------------------------------
	// verifica se cambio di direzione X/Y (cambio ruote)
	//----------------------------------------------------
	IF(auxSta.Stato_Aux_ASRV.Fermo_in_X = TRUE AND sP.Comandi.In_Mov_Y = TRUE) OR
	  (auxSta.Stato_Aux_ASRV.Fermo_in_Y = TRUE AND sP.Comandi.In_Mov_X = TRUE) THEN  
		bCambioDir := TRUE;	
	END_IF
	//-------------------------------------------------------------
	// Elabora solo se ASRV non è su Pintend oppure se non ho
	// il comando di Stop ASRV oppure trascorso Tmr cambio direzione
	//-------------------------------------------------------------
	bStop := FALSE;
	IF auxSta.Pos_ASRV = auxCmd.Pintend_PC OR auxCmd.Comando_PC.Stop = TRUE OR 
	   (bCambioDir = TRUE AND fbTCambioDir.Q = FALSE) THEN
		bStop := TRUE;
	END_IF
	IF bStop = FALSE THEN
		IF sP.Comandi.In_Mov_X THEN auxSta.Stato_ASRV.In_Mov_X := TRUE; END_IF
		IF sP.Comandi.In_Mov_Y THEN auxSta.Stato_ASRV.In_Mov_Y := TRUE; END_IF
		IF sP.Comandi.In_Mov_Av THEN auxSta.Stato_ASRV.In_Mov_Av := TRUE; END_IF
		IF sP.Comandi.In_Mov_Ind THEN auxSta.Stato_ASRV.In_Mov_Ind := TRUE; END_IF
		auxSta.Stato_Aux_ASRV.Fermo_in_X := FALSE;	
		auxSta.Stato_Aux_ASRV.Fermo_in_Y := FALSE;	
		bCambioDir := FALSE;	
		//----------------------------------------------------
		// Se Non nuovo Step incrementa offset + su Nodo=False 
		//----------------------------------------------------
		IF bSimRunNew=FALSE THEN 
			//----------------------------------------------------
			// Se abilitato Lenta allora incrementa solo 1 unità
			//----------------------------------------------------
			fCmSpost := fCmVel;
			IF sP.Comandi.Lenta = TRUE THEN
				fCmSpost := fCmLen;
			END_IF
			
			//######
			//------------------------------------------
			// Se cambio direzione step successivo allora
			// lenta con un pò di anticipo
			//------------------------------------------
			IF sP.Comandi.In_Mov_X <> sP_1.Comandi.In_Mov_X OR 
               sP.Comandi.In_Mov_Y <> sP_1.Comandi.In_Mov_Y THEN
				IF (auxSta.offset_da_nodo_ASRV+30 > sP.dist AND bRitroso=FALSE) OR 
				   (auxSta.offset_da_nodo_ASRV < 30 AND bRitroso=TRUE) THEN
					fCmSpost := fCmLen;
				END_IF 
			END_IF
			//######
			
			//---------------------------------------------------------------------------------------
			// Se Pos. attuale ASRV = Pos.Step allora ASRV decrementa distanza da Nodo. 
			// (sta ritornando su Nodo ingresso Magazzino)
			// UINT = 0..32767 positivo 32768..65xxx negativo
			//---------------------------------------------------------------------------------------
			IF bRitroso =TRUE THEN				        // movimento a ritroso
				IF auxSta.offset_da_nodo_ASRV>0 AND auxSta.offset_da_nodo_ASRV<=32767 THEN	        // decrementa solo se distanza >0
					auxSta.offset_da_nodo_ASRV := auxSta.offset_da_nodo_ASRV - TO_UINT(fCmSpost);	// si avvicina a nodo:  offset - X cm
					IF auxSta.offset_da_nodo_ASRV>32767 THEN   										// se negativo.. =0
						auxSta.offset_da_nodo_ASRV:=0;
					END_IF
				END_IF		
			ELSE
				auxSta.offset_da_nodo_ASRV := auxSta.offset_da_nodo_ASRV + TO_UINT(fCmSpost);		// si allontana da nodo: offset + X cm
			END_IF
			auxSta.Stato_ASRV.Su_Nodo := FALSE;														// Fuori nodo
			
			//------------------------------------------------------------
			// Verifica Distanza Percorsa >= Dist. Step. Se si nuovo Step
			//------------------------------------------------------------
			IF (auxSta.offset_da_nodo_ASRV >= sp.dist AND bRitroso=FALSE) OR	// Se avanti + offset >= distanza step
			   (auxSta.offset_da_nodo_ASRV <=0 AND bRitroso=TRUE)   THEN		// Se indietro + offset <= 0
							
				//§§§ 08/08/2022 - gestione carico/scarico con Offset
				bCS_Offset := FALSE;	// carico/scarico con offset
				//--------------------------------------------
				// Passo Carico con offset
				//--------------------------------------------
				IF sP.Comandi.CarSoll_0 OR
	   				sP.Comandi.CarSoll_1 THEN
					auxSta.Stato_ASRV.Carico := TRUE;
					auxSta.Peso_Teorico_ASRV := PESO_FITTIZIO_SIM;	// fittizio
					bCS_Offset := TRUE;	// carico/scarico con offset
					bCarSCar:=TRUE;		// Tmr  Carico/Scarico
				END_IF
				//--------------------------------------------
				// Passo Scarico con offset
				//--------------------------------------------
				IF sP.Comandi.Scarica THEN
					auxSta.Stato_ASRV.Carico := FALSE;
					auxSta.Peso_Teorico_ASRV := 0;	
					bCS_Offset := TRUE;	// carico/scarico con offset
					bCarSCar:=TRUE;		// Tmr  Carico/Scarico
				END_IF
				//§§§

				auxSta.Pos_ASRV := sP.ps;			// Pos. step
				//§§§ 08/08/2022 - gestione carico/scarico con Offset
				// Se carico/scarico con offset non azzera la distanza da nodo
				IF bCS_Offset= FALSE THEN
					auxSta.offset_da_nodo_ASRV := 0;	// offset = 0
					auxSta.Stato_ASRV.Su_Nodo := TRUE;	// Su nodo
				END_IF
				//§§§
				
				IF auxSta.Stato_ASRV.In_Mov_X = TRUE THEN
					auxSta.Stato_Aux_ASRV.Fermo_in_X := TRUE;	
				END_IF
				IF auxSta.Stato_ASRV.In_Mov_Y = TRUE THEN
					auxSta.Stato_Aux_ASRV.Fermo_in_Y := TRUE;	
				END_IF
				auxSta.Stato_ASRV.In_Mov_Av := FALSE;
				auxSta.Stato_ASRV.In_Mov_Ind := FALSE;
				auxSta.Stato_ASRV.In_Mov_X := FALSE;
				auxSta.Stato_ASRV.In_Mov_Y := FALSE;
				bSimRunNew := TRUE;
				//--------------------------------------------------
				// Se abilitato Step, mette in Hold la simulazione
				//--------------------------------------------------
				IF bSimulaStep=TRUE THEN
					bSimulaRun := FALSE;
				END_IF
			END_IF
		END_IF
	END_IF
END_IF

END_FUNCTION

// ---- POUs/Trasf_Sta_TxSta.TcPOU
FUNCTION Trasf_Sta_TxSta
VAR_INPUT
	auxSta   : REFERENCE TO STA_ASRV;
	auxTxSta : REFERENCE TO TX_STA_ASRV;
END_VAR
VAR
	ni : UINT :=0;
END_VAR

//-------------------------------------------------------------------
// Trasferisce Stato ASRV in Buffer Tx a PC
// Compatta le struttura Stato_ASRV (16 byte) in Word (16 bit)
// Stato ASRV --> STATO TX
//-------------------------------------------------------------------
auxTxSta.WatchDog_ASRV       := auxSta.WatchDog_ASRV;
auxTxSta.Pos_ASRV            := auxSta.Pos_ASRV;
auxTxSta.Stato_MIss_ASRV     := auxSta.Stato_MIss_ASRV;
auxTxSta.ptr_step_ASRV       := auxSta.ptr_step_ASRV;
auxTxSta.offset_da_nodo_ASRV := auxSta.offset_da_nodo_ASRV;
auxTxSta.Allarmi_1_ASRV      := auxSta.Allarmi_1_ASRV;
auxTxSta.Allarmi_2_ASRV      := auxSta.Allarmi_2_ASRV;
auxTxSta.Allarmi_3_ASRV      := auxSta.Allarmi_3_ASRV;
auxTxSta.Allarmi_4_ASRV      := auxSta.Allarmi_4_ASRV;
auxTxSta.Perc_Batteria_ASRV  := auxSta.Perc_Batteria_ASRV;
auxTxSta.Peso_Teorico_ASRV   := auxSta.Peso_Teorico_ASRV;
auxTxSta.StFree1             := auxSta.StFree1;
auxTxSta.StFree2             := auxSta.StFree2;
auxTxSta.StFree3             := auxSta.StFree3;
auxTxSta.StFree4             := auxSta.StFree4;
auxTxSta.StFree5             := auxSta.StFree5;
//------
auxTxSta.Stato_ASRV := BOOL_TO_UINT( auxSta.Stato_ASRV.In_Mov_X );
auxTxSta.Stato_ASRV := auxTxSta.Stato_ASRV + BOOL_TO_UINT( auxSta.Stato_ASRV.In_Mov_Y      ) * 2;
auxTxSta.Stato_ASRV := auxTxSta.Stato_ASRV + BOOL_TO_UINT( auxSta.Stato_ASRV.In_Mov_Av     ) * 4;
auxTxSta.Stato_ASRV := auxTxSta.Stato_ASRV + BOOL_TO_UINT( auxSta.Stato_ASRV.In_Mov_Ind    ) * 8;
auxTxSta.Stato_ASRV := auxTxSta.Stato_ASRV + BOOL_TO_UINT( auxSta.Stato_ASRV.In_Allarme    ) * 16;
auxTxSta.Stato_ASRV := auxTxSta.Stato_ASRV + BOOL_TO_UINT( auxSta.Stato_ASRV.Ok_Prog       ) * 32;
auxTxSta.Stato_ASRV := auxTxSta.Stato_ASRV + BOOL_TO_UINT( auxSta.Stato_ASRV.In_Automatico ) * 64;
auxTxSta.Stato_ASRV := auxTxSta.Stato_ASRV + BOOL_TO_UINT( auxSta.Stato_ASRV.In_Manuale    ) * 128;
auxTxSta.Stato_ASRV := auxTxSta.Stato_ASRV + BOOL_TO_UINT( auxSta.Stato_ASRV.Su_Nodo       ) * 256;
auxTxSta.Stato_ASRV := auxTxSta.Stato_ASRV + BOOL_TO_UINT( auxSta.Stato_ASRV.Carico        ) * 512;
auxTxSta.Stato_ASRV := auxTxSta.Stato_ASRV + BOOL_TO_UINT( auxSta.Stato_ASRV.PosSoll_0     ) * 1024;
auxTxSta.Stato_ASRV := auxTxSta.Stato_ASRV + BOOL_TO_UINT( auxSta.Stato_ASRV.PosSoll_1     ) * 2048;
auxTxSta.Stato_ASRV := auxTxSta.Stato_ASRV + BOOL_TO_UINT( auxSta.Stato_ASRV.Rich_Reset    ) * 4096;
auxTxSta.Stato_ASRV := auxTxSta.Stato_ASRV + BOOL_TO_UINT( auxSta.Stato_ASRV.Aux13         ) * 8192;
auxTxSta.Stato_ASRV := auxTxSta.Stato_ASRV + BOOL_TO_UINT( auxSta.Stato_ASRV.Aux14         ) * 16384;
auxTxSta.Stato_ASRV := auxTxSta.Stato_ASRV + BOOL_TO_UINT( auxSta.Stato_ASRV.Aux15         ) * 32768;
//------
auxTxSta.Stato_Aux_ASRV := BOOL_TO_UINT( auxSta.Stato_Aux_ASRV.Fermo_in_X );
auxTxSta.Stato_Aux_ASRV := auxTxSta.Stato_Aux_ASRV + BOOL_TO_UINT( auxSta.Stato_Aux_ASRV.Fermo_in_Y    ) * 2;
auxTxSta.Stato_Aux_ASRV := auxTxSta.Stato_Aux_ASRV + BOOL_TO_UINT( auxSta.Stato_Aux_ASRV.Rotaz_in_X    ) * 4;
auxTxSta.Stato_Aux_ASRV := auxTxSta.Stato_Aux_ASRV + BOOL_TO_UINT( auxSta.Stato_Aux_ASRV.Rotaz_in_Y    ) * 8;
auxTxSta.Stato_Aux_ASRV := auxTxSta.Stato_Aux_ASRV + BOOL_TO_UINT( auxSta.Stato_Aux_ASRV.In_Ricarica   ) * 16;
auxTxSta.Stato_Aux_ASRV := auxTxSta.Stato_Aux_ASRV + BOOL_TO_UINT( auxSta.Stato_Aux_ASRV.In_Sost_Batt  ) * 32;
auxTxSta.Stato_Aux_ASRV := auxTxSta.Stato_Aux_ASRV + BOOL_TO_UINT( auxSta.Stato_Aux_ASRV.In_Manutenz   ) * 64;
auxTxSta.Stato_Aux_ASRV := auxTxSta.Stato_Aux_ASRV + BOOL_TO_UINT( auxSta.Stato_Aux_ASRV.Aux7          ) * 128;
auxTxSta.Stato_Aux_ASRV := auxTxSta.Stato_Aux_ASRV + BOOL_TO_UINT( auxSta.Stato_Aux_ASRV.Aux8          ) * 256;
auxTxSta.Stato_Aux_ASRV := auxTxSta.Stato_Aux_ASRV + BOOL_TO_UINT( auxSta.Stato_Aux_ASRV.Aux9          ) * 512;
auxTxSta.Stato_Aux_ASRV := auxTxSta.Stato_Aux_ASRV + BOOL_TO_UINT( auxSta.Stato_Aux_ASRV.Aux10         ) * 1024;
auxTxSta.Stato_Aux_ASRV := auxTxSta.Stato_Aux_ASRV + BOOL_TO_UINT( auxSta.Stato_Aux_ASRV.Aux11         ) * 2048;
auxTxSta.Stato_Aux_ASRV := auxTxSta.Stato_Aux_ASRV + BOOL_TO_UINT( auxSta.Stato_Aux_ASRV.Aux12         ) * 4096;
auxTxSta.Stato_Aux_ASRV := auxTxSta.Stato_Aux_ASRV + BOOL_TO_UINT( auxSta.Stato_Aux_ASRV.Aux13         ) * 8192;
auxTxSta.Stato_Aux_ASRV := auxTxSta.Stato_Aux_ASRV + BOOL_TO_UINT( auxSta.Stato_Aux_ASRV.Aux14         ) * 16384;
auxTxSta.Stato_Aux_ASRV := auxTxSta.Stato_Aux_ASRV + BOOL_TO_UINT( auxSta.Stato_Aux_ASRV.Aux15         ) * 32768;

END_FUNCTION

// ---- POUs/FB_ClassASRV.TcPOU
FUNCTION_BLOCK PUBLIC FB_ClassASRV
VAR
	sAsrv 	 : 	ASRV;	// struttura ASRV	
END_VAR

METHOD PUBLIC Aggiorna_CMD_da_PC : BOOL
VAR_INPUT
	auxCmd   : REFERENCE TO CMD_PC;
END_VAR
//-------------------------------------
// Aggiorna struttura -> ASRV 1 - CMD  
//-------------------------------------
sAsrv.ASRV_CMD := auxCmd;
Aggiorna_CMD_da_PC := FALSE;	// errore
END_METHOD

METHOD PUBLIC Aggiorna_MIS_da_PC : BOOL
VAR_INPUT
	auxMis   : REFERENCE TO MIS_PC;
END_VAR
//------------------------------------
// Aggiorna struttura -> ASRV 1 - MIS 
//------------------------------------
sAsrv.ASRV_MIS := auxMis;
Aggiorna_MIS_da_PC := FALSE;	// errore
END_METHOD

METHOD PUBLIC Aggiorna_STA_a_PC : BOOL
VAR_INPUT
	auxSta   : REFERENCE TO STA_ASRV;
END_VAR
//-----------------------------------
// Aggiorna da struttura <- STA  
//----------------------------------
auxSta := sAsrv.ASRV_STA;
Aggiorna_STA_a_PC := FALSE;	// errore
END_METHOD

METHOD PUBLIC Azzera_MIS : BOOL
VAR
	ndim	: USINT;
	ni		: UINT; 	
END_VAR
//-------------------------------
// Azzera struttura -> MIS  
//-------------------------------
sAsrv.ASRV_MIS.Tot_step_PC   := 0;
sAsrv.ASRV_MIS.Pstart_PC     := 0;
sAsrv.ASRV_MIS.Pend_PC       := 0;
sAsrv.ASRV_MIS.Typ_car_PC    := 0;
sAsrv.ASRV_MIS.MisFree1      := 0;
sAsrv.ASRV_MIS.MisFree2      := 0;
sAsrv.ASRV_MIS.MisFree3      := 0;
//------------------------- Reset Step[]
FOR ni :=0 TO MAX_STEP_MISS BY 1 DO
	ndim := TO_USINT(SIZEOF(sAsrv.ASRV_MIS.Step_PC[ni]));							// dim. setp (short)
	MEMSET(destAddr:=ADR(sAsrv.ASRV_MIS.Step_PC[ni]) , fillByte:=ndim , n:=16#00 );	// max 255 byte!
END_FOR

//----------------------------
// Reset Step programma
//----------------------------
sAsrv.ASRV_STA.ptr_step_ASRV 	:=0;	// Reset puntatori Step
sAsrv.ASRV_STA.Stato_Miss_ASRV 	:=0;	// reset anche Stato Missione (anche se dovrebbe già essere 0)
//-------------------------------- memorizza stop su direzione X,Y
IF sAsrv.ASRV_STA.Stato_ASRV.In_Mov_X = TRUE THEN
	sAsrv.ASRV_STA.Stato_Aux_ASRV.Fermo_in_X := TRUE;	
END_IF
IF sAsrv.ASRV_STA.Stato_ASRV.In_Mov_Y = TRUE THEN
	sAsrv.ASRV_STA.Stato_Aux_ASRV.Fermo_in_Y := TRUE;	
END_IF
sAsrv.ASRV_STA.Stato_ASRV.In_Mov_Av := FALSE;
sAsrv.ASRV_STA.Stato_ASRV.In_Mov_Ind := FALSE;
sAsrv.ASRV_STA.Stato_ASRV.In_Mov_X   := FALSE;
sAsrv.ASRV_STA.Stato_ASRV.In_Mov_Y   := FALSE;
Azzera_MIS := FALSE;	// errore
END_METHOD

METHOD PUBLIC Get_sAsrv : BOOL
VAR_INPUT
	auxAsrv   : REFERENCE TO ASRV;
END_VAR
//------------------------------------------------------------------------------
// Recupera struttura globale "sAsrv" di Classe >> struttura locale di appoggio
//-------------------------------------------------------------------------------
auxAsrv := sAsrv;
END_METHOD

METHOD PUBLIC Set_sAsrv : BOOL
VAR_INPUT
	auxAsrv   : REFERENCE TO ASRV;
END_VAR
//------------------------------------------------------------------------------
// Salva struttura locale di appoggio >> struttura globale di Classe "sAsrv" 
//-------------------------------------------------------------------------------
sAsrv := auxAsrv;
END_METHOD

END_FUNCTION_BLOCK

// ---- POUs/FB_Test_XXX.TcPOU
FUNCTION_BLOCK FB_Test_XXX
VAR_INPUT
	TestMisPOINT_XXX : POINTER TO MIS_PC;	// Passaggio tramite Pointer
	TestMisREFER_XXX : POINTER TO MIS_PC;	// Passaggio tramite Reference
	
END_VAR

// Lo scopo di questa FB è verificare come passare dei parametri all'interno della FB utilizzando 
// VAR_INPUT. In pratica passiamo un puntatore ad una struttra di tipo MIS_PC
// All'interno della funzione poi per accedere agli elementi della strutttura passata come puntatore, utilizziamo ^" 

TestMisPOINT_XXX^.Pend_PC := 100;
TestMisPOINT_XXX^.Pstart_PC := 10;

TestMisREFER_XXX^.Pend_PC :=20;

END_FUNCTION_BLOCK

// ---- GlobalTextList.TcGTLO
TEXTLIST GlobalTextList
  422 = '%04x'
  486 = '%4x'
  277 = '%d'
  672 = '%d  Kg'
  179 = '%d %%'
  341 = 'Allarmi_1_ASRV'
  516 = 'Allarmi_1_ASRV (hex)'
  278 = 'Allarmi_2_ASRV'
  317 = 'Allarmi_2_ASRV (hex)'
  303 = 'Allarmi_3_ASRV'
  767 = 'Allarmi_3_ASRV (hex)'
  573 = 'Allarmi_4_ASRV'
  605 = 'Allarmi_4_ASRV (hex)'
  759 = 'Aux13'
  85 = 'Aux14'
  645 = 'Aux15'
  844 = 'Cambio direzione'
  282 = 'Carico'
  402 = 'CarSoll_0'
  577 = 'CarSoll_1'
  938 = 'CmFree1'
  294 = 'Comandi PC'
  43 = 'dist'
  867 = 'dist (distanza)'
  743 = 'End'
  413 = 'End_Miss_PC'
  292 = 'Errore Comunicaz.'
  432 = 'Errore Comunicaz. PC'
  877 = 'Errore Comunicazione'
  471 = 'Errore Comunicazione PC'
  339 = 'Fermo_in_X'
  989 = 'Fermo_in_Y'
  519 = 'Hold Simulazione'
  751 = 'Inching (Hold a fine Step)'
  827 = 'In_Allarme'
  886 = 'In_Automatico'
  876 = 'In_Manuale'
  495 = 'In_Mov_Av'
  687 = 'In_Mov_Ind'
  647 = 'In_Mov_X'
  152 = 'In_Mov_Y'
  520 = 'In_Ricarica'
  435 = 'Lenta'
  245 = 'New_Pos_PC'
  515 = 'offset_da_Nodo_ASRV'
  836 = 'Ok_Progr'
  873 = 'Pend_PC'
  612 = 'Perc_Batteria_ASRV'
  353 = 'Peso_Teorico_ASRV'
  842 = 'Pintend_PC'
  975 = 'PosSoll_0'
  696 = 'PosSoll_1'
  158 = 'Pos_ASRV'
  295 = 'ps'
  104 = 'ps (nodo)'
  782 = 'Pstart_PC'
  828 = 'ptr_step_ASRV'
  653 = 'rall'
  629 = 'Rapp. Veloce / Lenta'
  470 = 'Rich_Reset'
  288 = 'Run'
  382 = 'Run / Hold'
  968 = 'Scarica'
  118 = 'Simulatore Veicolo ASRV'
  478 = 'Simulatore Veicolo ASRV (v.0.1)'
  431 = 'Simulazione RUN '
  472 = 'sRxCmd.WatchDog_PC'
  840 = 'Start_Miss_PC'
  766 = 'Stato ASRV '
  547 = 'Stato_Miss_ASRV'
  465 = 'Step'
  620 = 'Step 1'
  923 = 'Step by Step'
  313 = 'Step Missione'
  681 = 'Stop'
  91 = 'Su_Nodo'
  732 = 'Tmr Cambio direz.'
  988 = 'Tmr Cambio direzione'
  536 = 'Tmr Carico/Scarico'
  102 = 'Tot_Step_PC'
  426 = 'TO_STRING(sRxCmd.WatchDog_PC)'
  121 = 'Typ_Car_PC'
  969 = 'V.1.0'
  506 = 'V.1.1'
  582 = 'V.1.2'
  226 = 'Vel. Simulaz. (cm 1/10s)'
  270 = 'Vel. Simulazione (cm 1/10s)'
  304 = 'Velocità Sim.'
  75 = 'Velocità Sim. (cm/clock)'
  275 = 'Velocità Simulaz.'
  35 = 'Velocità Simulaz. (cm 1/10s)'
  125 = 'Velocità Simulazione'
  563 = 'WatchDog ASRV: %d'
  761 = 'WatchDog PC: %d'
  795 = 'WatchDog_ASRV'
  29 = 'WatchDog_PC'
END_TEXTLIST

// ---- VISUs/Visualization.TcVIS
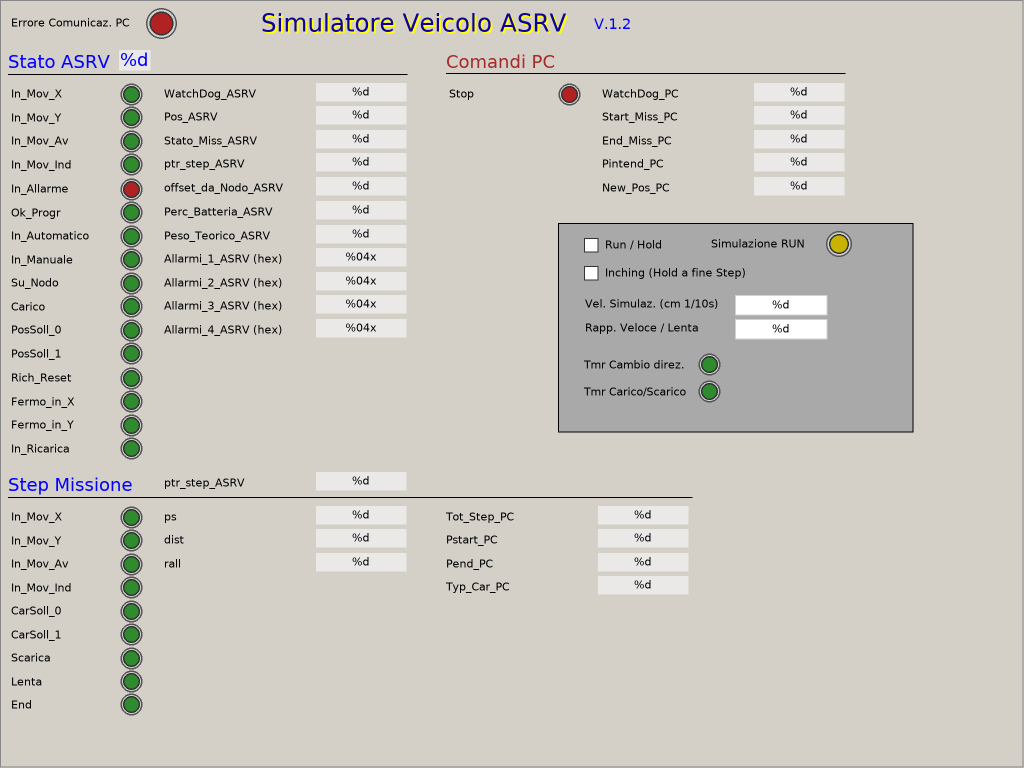
VISUALIZATION Visualization  // 1024x768
    Rectangle (558,223 355x209)
    Label (8,79 113x30), "In_Mov_X"
    Label (8,103 113x30), "In_Mov_Y"
    Lamp1 (119,82 25x25), variable: sSta.Stato_ASRV.In_Mov_X, style: Lamp-Lamp1-Green
    Lamp1 (119,105 25x25), variable: sSta.Stato_ASRV.In_Mov_Y, style: Lamp-Lamp1-Green
    Label (8,126 113x30), "In_Mov_Av"
    Label (8,150 113x30), "In_Mov_Ind"
    Lamp1 (119,129 25x25), variable: sSta.Stato_ASRV.In_Mov_Av, style: Lamp-Lamp1-Green
    Lamp1 (119,152 25x25), variable: sSta.Stato_ASRV.In_Mov_Ind, style: Lamp-Lamp1-Green
    Label (8,174 113x30), "In_Allarme"
    Label (8,198 113x30), "Ok_Progr"
    Lamp1 (119,177 25x25), variable: sSta.Stato_ASRV.In_Allarme, style: Lamp-Lamp1-Red
    Lamp1 (119,200 25x25), variable: sSta.Stato_ASRV.Ok_Prog, style: Lamp-Lamp1-Green
    Label (8,221 113x30), "In_Automatico"
    Label (8,245 113x30), "In_Manuale"
    Lamp1 (119,224 25x25), variable: sSta.Stato_ASRV.In_Automatico, style: Lamp-Lamp1-Green
    Lamp1 (119,247 25x25), variable: sSta.Stato_ASRV.In_Manuale, style: Lamp-Lamp1-Green
    Label (8,268 113x30), "Su_Nodo"
    Label (8,292 113x30), "Carico"
    Lamp1 (119,271 25x25), variable: sSta.Stato_ASRV.Su_Nodo, style: Lamp-Lamp1-Green
    Lamp1 (119,294 25x25), variable: sSta.Stato_ASRV.Carico, style: Lamp-Lamp1-Green
    Label (8,315 113x30), "PosSoll_0"
    Label (8,339 113x30), "PosSoll_1"
    Lamp1 (119,318 25x25), variable: sSta.Stato_ASRV.PosSoll_0, style: Lamp-Lamp1-Green
    Lamp1 (119,341 25x25), variable: sSta.Stato_ASRV.PosSoll_1, style: Lamp-Lamp1-Green
    Label (8,363 113x30), "Rich_Reset"
    Label (8,387 113x30), "Fermo_in_X"
    Lamp1 (119,366 25x25), variable: sSta.Stato_ASRV.Rich_Reset, style: Lamp-Lamp1-Green
    Lamp1 (119,389 25x25), variable: sSta.Stato_Aux_ASRV.Fermo_in_X, style: Lamp-Lamp1-Green
    Label (8,410 113x30), "Fermo_in_Y"
    Label (8,434 113x30), "In_Ricarica"
    Lamp1 (119,413 25x25), variable: sSta.Stato_Aux_ASRV.Fermo_in_Y, style: Lamp-Lamp1-Green
    Lamp1 (119,436 25x25), variable: sSta.Stato_Aux_ASRV.In_Ricarica, style: Lamp-Lamp1-Green
    Label (8,8 132x30), "Errore Comunicaz. PC"
    Lamp1 (144,6 35x35), variable: bErrComPc, style: Lamp-Lamp1-Red
    Label (5,47 143x30), "Stato ASRV"
    Label (161,102 130x30), "Pos_ASRV"
    Label (161,126 130x30), "Stato_Miss_ASRV"
    Label (161,149 130x30), "ptr_step_ASRV"
    Label (161,173 130x30), "offset_da_Nodo_ASRV"
    Label (161,197 130x30), "Perc_Batteria_ASRV"
    Label (161,221 130x30), "Peso_Teorico_ASRV"
    Label (161,244 130x30), "Allarmi_1_ASRV (hex)"
    Label (161,268 130x30), "Allarmi_2_ASRV (hex)"
    Label (161,291 130x30), "Allarmi_3_ASRV (hex)"
    Label (161,315 130x30), "Allarmi_4_ASRV (hex)"
    Textfield (315,105 92x20), "%d", text variable: sTxSta.Pos_ASRV
    Textfield (315,129 92x20), "%d", text variable: sTxSta.Stato_Miss_ASRV
    Textfield (315,152 92x20), "%d", text variable: sTxSta.ptr_step_ASRV
    Textfield (315,176 92x20), "%d", text variable: sTxSta.offset_da_nodo_ASRV
    Textfield (315,200 92x20), "%d", text variable: sTxSta.Perc_Batteria_ASRV
    Textfield (315,224 92x20), "%d", text variable: sTxSta.Peso_Teorico_ASRV
    Textfield (315,247 92x20), "%04x", text variable: sTxSta.Allarmi_1_ASRV
    Textfield (315,271 92x20), "%04x", text variable: sTxSta.Allarmi_2_ASRV
    Textfield (315,294 92x20), "%04x", text variable: sTxSta.Allarmi_3_ASRV
    Textfield (315,318 92x20), "%04x", text variable: sTxSta.Allarmi_4_ASRV
    Label (161,79 130x30), "WatchDog_ASRV"
    Textfield (315,82 92x20), "%d", text variable: sTxSta.WatchDog_ASRV
    Label (446,79 113x30), "Stop"
    Lamp1 (557,82 25x25), variable: fbClassAsrv.sAsrv.ASRV_CMD.Comando_PC.Stop, style: Lamp-Lamp1-Red
    Label (443,47 143x30), "Comandi PC"
    Label (599,102 130x30), "Start_Miss_PC"
    Label (599,126 130x30), "End_Miss_PC"
    Label (599,149 130x30), "Pintend_PC"
    Label (599,173 130x30), "New_Pos_PC"
    Textfield (753,105 92x20), "%d", text variable: sRxCmd.Start_Miss_PC
    Textfield (753,129 92x20), "%d", text variable: sRxCmd.End_Miss_PC
    Textfield (753,152 92x20), "%d", text variable: sRxCmd.Pintend_PC
    Textfield (753,176 92x20), "%d", text variable: sRxCmd.New_Pos_PC
    Label (599,79 130x30), "WatchDog_PC"
    Textfield (753,82 92x20), "%d", text variable: sRxCmd.WatchDog_PC
    Line (8,74) (407,74)
    Line (446,73) (845,73)
    Label (8,502 113x30), "In_Mov_X"
    Label (8,526 113x30), "In_Mov_Y"
    Lamp1 (119,505 25x25), variable: sLastStep.Comandi.In_Mov_X, style: Lamp-Lamp1-Green
    Lamp1 (119,528 25x25), variable: sLastStep.Comandi.In_Mov_Y, style: Lamp-Lamp1-Green
    Label (8,549 113x30), "In_Mov_Av"
    Label (8,573 113x30), "In_Mov_Ind"
    Lamp1 (119,552 25x25), variable: sLastStep.Comandi.In_Mov_Av, style: Lamp-Lamp1-Green
    Lamp1 (119,575 25x25), variable: sLastStep.Comandi.In_Mov_Ind, style: Lamp-Lamp1-Green
    Label (5,470 143x30), "Step Missione"
    Label (161,525 130x30), "dist"
    Label (161,549 130x30), "rall"
    Textfield (315,528 92x20), "%d", text variable: sLastStep.dist
    Textfield (315,552 92x20), "%d", text variable: sLastStep.rall
    Label (161,502 130x30), "ps"
    Textfield (315,505 92x20), "%d", text variable: sLastStep.ps
    Line (8,497) (692,497)
    Label (8,596 113x30), "CarSoll_0"
    Label (8,620 113x30), "CarSoll_1"
    Lamp1 (119,599 25x25), variable: sLastStep.Comandi.CarSoll_0, style: Lamp-Lamp1-Green
    Lamp1 (119,622 25x25), variable: sLastStep.Comandi.CarSoll_1, style: Lamp-Lamp1-Green
    Label (8,643 113x30), "Scarica"
    Label (8,667 113x30), "Lenta"
    Lamp1 (119,646 25x25), variable: sLastStep.Comandi.Scarica, style: Lamp-Lamp1-Green
    Lamp1 (119,669 25x25), variable: sLastStep.Comandi.Lenta, style: Lamp-Lamp1-Green
    Label (161,468 130x30), "ptr_step_ASRV"
    Textfield (315,471 92x20), "%d", text variable: sTxSta.ptr_step_ASRV
    Label (8,690 113x30), "End"
    Lamp1 (119,692 25x25), variable: sLastStep.Comandi.End, style: Lamp-Lamp1-Green
    Label (443,525 130x30), "Pstart_PC"
    Label (443,549 130x30), "Pend_PC"
    Label (443,572 130x30), "Typ_Car_PC"
    Textfield (597,528 92x20), "%d", text variable: fbClassAsrv.sAsrv.ASRV_MIS.Pstart_PC
    Textfield (597,552 92x20), "%d", text variable: fbClassAsrv.sAsrv.ASRV_MIS.Pend_PC
    Textfield (597,575 92x20), "%d", text variable: fbClassAsrv.sAsrv.ASRV_MIS.Typ_car_PC
    Label (443,502 130x30), "Tot_Step_PC"
    Textfield (597,505 92x20), "%d", text variable: fbClassAsrv.sAsrv.ASRV_MIS.Tot_step_PC
    Textfield (118,49 33x22), "%d", text variable: fbClassAsrv.sAsrv.ASRV_num
    Label (582,289 150x30), "Vel. Simulaz. (cm 1/10s)"
    Textfield (735,295 92x20), "%d", text variable: nSimCmSpost
        OnMouseClick: write the text variable via VisuDialogs.Numpad, min 1, max 100
    Label (582,313 150x30), "Rapp. Veloce / Lenta"
    Textfield (735,319 92x20), "%d", text variable: nRappVelLen
        OnMouseClick: write the text variable via VisuDialogs.Numpad, min 1, max 20
    Label (708,229 113x30), "Simulazione RUN"
    Lamp1 (824,229 30x30), variable: bSimulaRun, style: Lamp-Lamp1-Yellow
    Label (581,350 113x30), "Tmr Cambio direz."
    Lamp1 (697,352 25x25), variable: bCambioDir, style: Lamp-Lamp1-Green
    Label (260,10 330x30), "Simulatore Veicolo ASRV"
    Label (258,8 330x30), "Simulatore Veicolo ASRV"
    Label (591,9 49x30), "V.1.2"
    Checkbox (582,230 103x30), "Run / Hold", variable: bSimulaRun
    Checkbox (582,258 201x30), "Inching (Hold a fine Step)", variable: bSimulaStep
    Label (581,377 113x30), "Tmr Carico/Scarico"
    Lamp1 (697,379 25x25), variable: bCarScar, style: Lamp-Lamp1-Green
END_VISUALIZATION
